# EPICS autosave request: CARSApp/Db/auto_shutter_settings.req
$(P)$(SHUT)AutoOpenMode
$(P)$(SHUT)AutoOpenPeriod.DLY1
